Staubli VAL3: Simulation.pjx

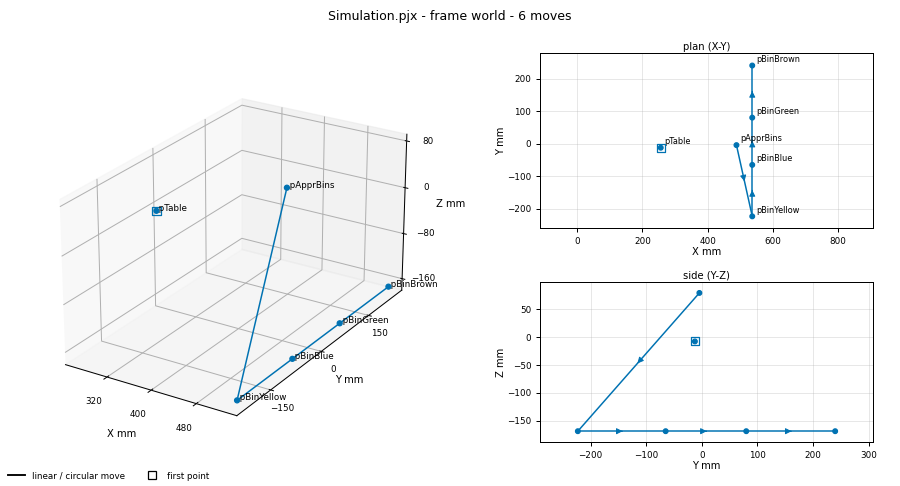
[picture p0: tool path of Simulation.pjx in frame world, 6 of 10 moves have a stored position in this frame; points joined in program order, loops and branches not executed]
--- Simulation.pjx ---
Parameters version=s7.11.2 stackSize=5000 millimeterUnit=true
Program file=moveRobot.pgx
Program file=pantalla.pgx
Program file=start.pgx
Program file=startingSockets.pgx
Program file=statesRobot.pgx
Program file=stop.pgx
Data file=Simulation.dtx

--- Simulation.dtx ---
mdesc mNomSpeed
sio sSocket = {link=Socket\Feedback}
tool tToolSuccion = {z=110, fatherId=flange[0], ioLink=valve2}
num nConnection
num nRecvData
jointRx JApproach1 = {j2=9, j3=75, j5=93}
jointRx JHome = {j3=0.6}
screen sMonitor
num l_nRetVal
pointRx pApprBins = {x=488.533117374584, y=-4.31537939334066, z=79.7509349968276, rx=-179.999994995315, ry=-0.671274884561614, rz=0.0461961759228383, fatherId=world[0]}
pointRx pBinYellow = {x=537, y=-223, z=-169, ry=-180, rz=78, fatherId=world[0]}
pointRx pBinBlue = {x=537, y=-65, z=-169, ry=-180, rz=78, fatherId=world[0]}
pointRx pBinGreen = {x=537, y=80, z=-169, ry=-180, rz=78, fatherId=world[0]}
pointRx pBinBrown = {x=537, y=240, z=-169, ry=-180, rz=78, fatherId=world[0]}
jointRx jGetCinta = {j1=-85, j2=70, j3=55, j5=56}
bool bStop
num nkey
jointRx jAproachCinta = {j1=-82, j2=60, j3=56.5, j5=65}
pointRx pTable = {x=256.13, y=-12.37, z=-7.47, ry=-180, rz=0.046191606806918, fatherId=world[0]}
tool tToolGripper = {z=115, fatherId=flange[0], ioLink=valve1}
sio sPlc = {link=Socket\PLClient}
num nRecvPLC

--- start.pgx ---
program start()
begin
  call startingSockets()
  taskCreate "stateRobot", 1, statesRobot()
  taskCreate "moveRobot", 1, moveRobot()
  taskCreate "screen", 1, pantalla()
end

--- MoveRobot.pgx ---
program moveRobot()
begin
  movej(JHome,tToolSuccion, mNomSpeed)
  waitEndMove()
  movej(JApproach1,tToolSuccion, mNomSpeed)
  waitEndMove()
  do
    movel(pTable,tToolSuccion, mNomSpeed)
    waitEndMove()
    sioGet(sPlc, nRecvPLC)
    if nRecvPLC == 100
      sioSet(sSocket, 82)
      movej(jAproachCinta, tToolSuccion, mNomSpeed)
      waitEndMove()
      movej(jGetCinta, tToolSuccion, mNomSpeed)
      waitEndMove()
      close(tToolSuccion)
      waitEndMove()
      movel(pApprBins, tToolSuccion, mNomSpeed)
      waitEndMove()
      nConnection = sioGet(sSocket, nRecvData)
    switch nRecvData
      case 48
        movel(pBinYellow, tToolSuccion, mNomSpeed)
        waitEndMove()
      break
      case 49
        movel(pBinBlue, tToolSuccion, mNomSpeed)
        waitEndMove()
      break
      case 50
        movel(pBinGreen, tToolSuccion, mNomSpeed)
        waitEndMove()
      break
      case 51
        movel(pBinBrown, tToolSuccion, mNomSpeed)
        waitEndMove()
      break
      default
        putln("Bin selected no correct")
      break
    endSwitch
      open(tToolSuccion)
      waitEndMove()
    endIf
  until 1==2
end

--- pantalla.pgx ---
program pantalla()
begin
  userPage(sMonitor)
  cls(sMonitor)
  title(sMonitor, "Start to recicling")
  gotoxy(sMonitor, 35,13)
  put(sMonitor, "EXIT")
  do
    gotoxy(sMonitor, 0,1)
    put(sMonitor, "Port 1102:")
    gotoxy(sMonitor, 12,1)
    switch nConnection
      case -1
        put(sMonitor, "Waiting connection")
      break
      case 1
        put(sMonitor, "Connected succesful")
        putln(sMonitor,"Go to bin: ")
        switch nRecvData
          case 48
            put(sMonitor, "Yellow")
          break
          case 49
           put(sMonitor, "Blue")
          break
        case 50
          put(sMonitor, "Green")
        break
        case 51
          put(sMonitor, "Brown")
        break
        default
          putln(sMonitor, "Bin selected no correct")
        break
      endSwitch
      break
      default
        put(sMonitor, "Connection lose")
      break
    endSwitch
  until 1==1
end

--- startingSockets.pgx ---
program startingSockets()
begin
  clearBuffer(sSocket)
  //clearBuffer(sPlc)
  wait(sioSet(sSocket, 73)==1)
  //wait(sioGet(sPlc, nRecvPLC)==1)
end

--- statesRobot.pgx ---
program statesRobot()
begin
  bStop = false
  do
    nkey = getKey()
    if(nkey == 278)
      bStop = true
      userPage()
      cls()
      gotoxy(14,6)
      put("FINAL PROGRAM")
      taskKill("moveRobot")
      taskKill("screen")
      taskKill("obatinValues")
      wait(taskStatus("moveRobot") == -1)
      wait(taskStatus("screen") == -1)
      wait(taskStatus("obatinValues") == -1)
    endIf
  until bStop == true


end
